TEXTLIST EL1809_M_2
  1 = 'Lower limit S1_8 ' | chinese: '压辊S1下限位8' | Chinese: '压辊S1下限位8'
  2 = 'Lower limit S1_9 ' | chinese: '压辊S1下限位9' | Chinese: '压辊S1下限位9'
  3 = 'Lower limit S1_10 ' | chinese: '压辊S1下限位10' | Chinese: '压辊S1下限位10'
  4 = 'Lower limit S1_11 ' | chinese: '压辊S1下限位11' | Chinese: '压辊S1下限位11'
  5 = 'Lower limit S1_12 ' | chinese: '压辊S1下限位12' | Chinese: '压辊S1下限位12'
  6 = 'Lower limit S1_13 ' | chinese: '压辊S1下限位13' | Chinese: '压辊S1下限位13'
  7 = 'Lower limit S1_14 ' | chinese: '压辊S1下限位14' | Chinese: '压辊S1下限位14'
  8 = 'Lower limit S1_15 ' | chinese: '压辊S1下限位15' | Chinese: '压辊S1下限位15'
  9 = 'Lower limit S1_16 ' | chinese: '压辊S1下限位16' | Chinese: '压辊S1下限位16'
  10 = 'L_front foot pedal1' | chinese: '左前脚踏开关1' | Chinese: '左前脚踏开关1'
  11 = 'L_front foot pedal2' | chinese: '左前脚踏开关2' | Chinese: '左前脚踏开关2'
  12 = 'L_front foot pedal3' | chinese: '左前脚踏开关3' | Chinese: '左前脚踏开关3'
  13 = 'R_front foot pedal1' | chinese: '右前脚踏开关1' | Chinese: '右前脚踏开关1'
  14 = 'R_front foot pedal2' | chinese: '右前脚踏开关2' | Chinese: '右前脚踏开关2'
  15 = 'R_front foot pedal3' | chinese: '右前脚踏开关3' | Chinese: '右前脚踏开关3'
  16 = 'L_rear foot pedal1' | chinese: '左后脚踏开关1' | Chinese: '左后脚踏开关1'
   = ''
END_TEXTLIST

(* stored: Version 1.1.0.1, ProductVersion 3.1.4024.11
   TextList EL1809_M_2: Id {96a655e3-2e1c-4a20-9058-28d27a9236c2} *)
